FUNCTION_BLOCK FB_BatteryConditioningSFC
VAR_IN_OUT
	IPSDemand					:	ST_PowerDemand;
	ConditioningRequirements	: 	ST_ConditioningRequirements;
	Control						:	ST_CoolingSystem_Control;
	Get							:	ST_CoolingSystemGet;	
END_VAR



VAR_OUTPUT
	SFCCurrentStep	:	STRING;
END_VAR
VAR_OUTPUT
	SFCActive	:	BOOL;
END_VAR

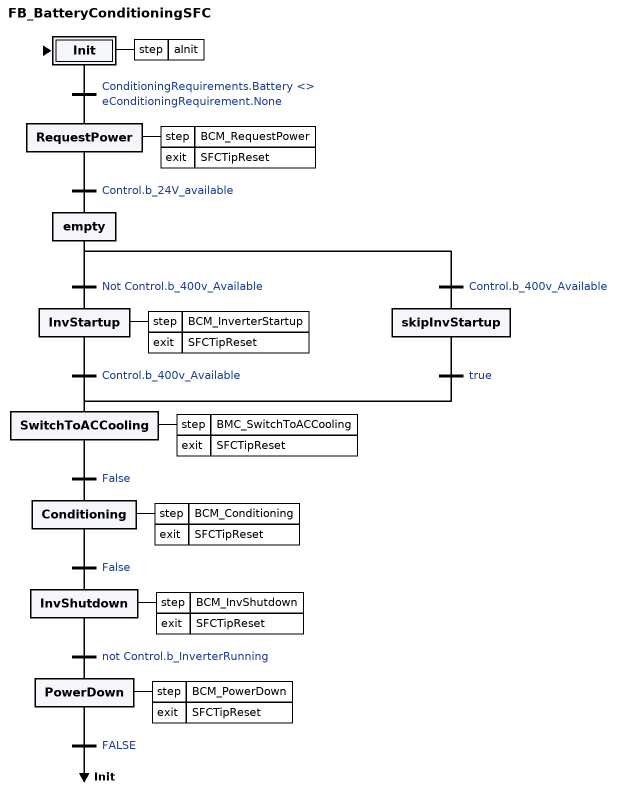
INITIAL_STEP Init:
    aInit(N);  // step action
END_STEP
TRANSITION FROM Init TO RequestPower
    := ConditioningRequirements.Battery <> eConditioningRequirement.None;
END_TRANSITION
STEP RequestPower:
    BCM_RequestPower(N);  // step action
    SFCTipReset(P0);  // exit action
END_STEP
TRANSITION FROM RequestPower TO empty
    := Control.b_24V_available;
END_TRANSITION
STEP empty:
END_STEP
TRANSITION FROM empty TO InvStartup
    := Not Control.b_400v_Available;
END_TRANSITION
STEP InvStartup:
    BCM_InverterStartup(N);  // step action
    SFCTipReset(P0);  // exit action
END_STEP
TRANSITION FROM InvStartup TO SwitchToACCooling
    := Control.b_400v_Available;
END_TRANSITION
TRANSITION FROM empty TO skipInvStartup
    := Control.b_400v_Available;
END_TRANSITION
STEP skipInvStartup:
END_STEP
TRANSITION FROM skipInvStartup TO SwitchToACCooling
    := true;
END_TRANSITION
STEP SwitchToACCooling:
    BMC_SwitchToACCooling(N);  // step action
    SFCTipReset(P0);  // exit action
END_STEP
TRANSITION FROM SwitchToACCooling TO Conditioning
    := False;
END_TRANSITION
STEP Conditioning:
    BCM_Conditioning(N);  // step action
    SFCTipReset(P0);  // exit action
END_STEP
TRANSITION FROM Conditioning TO InvShutdown
    := False;
END_TRANSITION
STEP InvShutdown:
    BCM_InvShutdown(N);  // step action
    SFCTipReset(P0);  // exit action
END_STEP
TRANSITION FROM InvShutdown TO PowerDown
    := not Control.b_InverterRunning;
END_TRANSITION
STEP PowerDown:
    BCM_PowerDown(N);  // step action
    SFCTipReset(P0);  // exit action
END_STEP
TRANSITION FROM PowerDown TO Init
    := FALSE;
END_TRANSITION

ACTION aInit:
SFCActive := False;
END_ACTION

ACTION BCM_Conditioning:

//No real demand for complicated regulation?
//system is off. Just return the average battery temperature to nominal.

//for now just test with fixed setpoints

CASE ConditioningRequirements.Battery OF
	eConditioningRequirement.Cooling:
		Control.e_HeatpumpMode := eHeatpumpmode.Cooling;
		Control.r_HeatPumpSetpoint := 15.0;//minimum adviced battery temperature. Setpoint could be lower, but watch out for inverter condensation.
	eConditioningRequirement.Heating:
		Control.e_HeatpumpMode := eHeatpumpmode.Heating;
		Control.r_HeatPumpSetpoint := 35.0; //minimum heating setpoint
	eConditioningRequirement.None:
		Control.e_HeatpumpMode := eHeatpumpmode.Standby;
		SFCTip := TRUE;
END_CASE

//if coolantpressure drops below startup minimum while inverter is running, shutdown system immediately!
IF 	Control.b_InverterRunning AND
 	(Control.r_CoolantPressure < (CoolingSystemParams.StartupPumpMinimumPressure + Control.r_CoolantIdlePressure)) THEN
		get.Events.b_InverterCoolingLoopError := TRUE;
		ConditioningRequirements.by_PSCoolingPowerMode := 0;
END_IF
END_ACTION

ACTION BCM_Cooldown:

IF ConditioningRequirements.Battery = eConditioningRequirement.Cooling THEN
	Control.b_CloseBatteryLoopValve := FALSE;
	Control.r_HeatPumpSetpoint := 15.0;
ELSIF ConditioningRequirements.Battery = eConditioningRequirement.Heating THEN
	Control.b_CloseBatteryLoopValve := FALSE;
	Control.r_HeatPumpSetpoint := 25.0;
ELSE
	//battery conditioning done, close valve to speed up other conditioning loops
	Control.b_CloseBatteryLoopValve := TRUE;
	IF ConditioningRequirements.Enclosure = eConditioningRequirement.Heating THEN
		Control.r_HeatPumpSetpoint := 25.0;
	ELSIF ConditioningRequirements.Enclosure = eConditioningRequirement.Cooling THEN
		Control.r_HeatPumpSetpoint := 15.0;
	//ELSE
		//if enclosure and battery are ok. Inverter is presumably already cooled down enough. 
		//If not, keep running in current mode for longer
	//	IF PSGet.r_TemperatureMax < CoolingSystemParams.InverterIdleShutdownTemp THEN
		//	ConditioningModeRequired := eConditioningStates.OFF;
		//END_IF
	END_IF	
END_IF
END_ACTION

ACTION BCM_InverterStartup:
Control.b_CloseBatteryLoopValve 	:= TRUE;
Control.b_CloseFancoilLoopValve		:= TRUE;
Control.b_CloseInverterLoopValve	:= FALSE;

Control.b_DCFancoilEnable	:=	FALSE;
//Control.b_ACFancoilEnable	:=	FALSE;

Control.b_DCPumpEnable		:= TRUE;
Control.b_ACPumpEnable		:= FALSE;

Control.b_HeatPumpPowerEnable := FALSE;

//if both are ok, the inverter should have enough flow to start
IF Control.r_CoolantPressure > (CoolingSystemParams.StartupPumpMinimumPressure + Control.r_CoolantIdlePressure) AND Control.b_InverterLoopEnabled THEN
	//Inverter may commence modulating, but no power delivery yet.
	ConditioningRequirements.by_PSCoolingPowerMode := 1;
END_IF
END_ACTION

ACTION BCM_InvShutdown:
Control.b_CloseBatteryLoopValve 	:= TRUE;
Control.b_CloseFancoilLoopValve	:= TRUE;
Control.b_CloseInverterLoopValve	:= FALSE;

Control.b_DCFancoilEnable	:=	FALSE;
//Control.b_ACFancoilEnable	:=	FALSE;

Control.b_DCPumpEnable		:= TRUE;
Control.b_ACPumpEnable		:= FALSE;

Control.b_HeatPumpPowerEnable := FALSE;

//Inverter may shutdown now
ConditioningRequirements.by_PSCoolingPowerMode := 0;
END_ACTION

ACTION BCM_PowerDown:
Control.b_CloseBatteryLoopValve 	:= 	FALSE;
Control.b_CloseFancoilLoopValve	:= 	FALSE;
Control.b_CloseInverterLoopValve	:= 	FALSE;

Control.b_DCFancoilEnable		:=	FALSE;
//Control.b_ACFancoilEnable		:=	FALSE;

Control.b_DCPumpEnable			:= 	FALSE;
Control.b_ACPumpEnable			:= 	FALSE;

Control.b_HeatPumpPowerEnable 	:= 	FALSE;

IPSDemand.b_Demand_24V 			:= FALSE;

Control.e_HeatpumpMode := eHeatpumpMode.Standby; 
SFCActive:= False;
END_ACTION

ACTION BCM_RequestPower:
SFCActive:= True;
IPSDemand.b_Demand_24V := TRUE;
IPSDemand.b_Demand_400V := TRUE;
END_ACTION

ACTION BMC_SwitchToACCooling:
Control.b_DCFancoilEnable 		:= FALSE;
//Control.b_ACFancoilEnable		:= FALSE;


//First enable both pumps to see if AC pump works (by checking pressure increase)
Control.b_ACPumpEnable 			:= TRUE;
Control.b_DCPumpEnable 			:= TRUE;

IF Control.r_CoolantPressure > (CoolingSystemParams.MainPumpMinimumPressure + Control.r_CoolantIdlePressure) THEN
	Control.b_CloseBatteryLoopValve 	:= FALSE;
	Control.b_CloseFancoilLoopValve 	:= FALSE;
	Control.b_CloseBatteryLoopValve 	:= FALSE;
	Control.b_HeatPumpPowerEnable 	:= TRUE;
	Control.b_DCPumpEnable 			:= FALSE;
	Control.e_HeatpumpMode := eHeatpumpmode.Standby;
	Control.r_HeatPumpSetpoint := 18.0;
	SFCTip := TRUE;
END_IF
END_ACTION

METHOD SFCEnable : BOOL
VAR_INPUT
	Enable	:	Bool;
END_VAR
IF Enable THEN
	SFCInit := FALSE;
ELSE
	SFCActive:= FALSE;
	SFCInit := TRUE;
END_IF
END_METHOD

ACTION SFCTipReset:
SFCTip := FALSE;
END_ACTION

END_FUNCTION_BLOCK

(* stored: Version 1.1.0.1, ProductVersion 3.1.4024.12
   POU FB_BatteryConditioningSFC: Id {5ce527d0-615b-41eb-9af7-e543097ab227}, SpecialFunc None
   Action aInit: Id {07ac61e1-8ac9-4677-8bb9-bcdeccba797d}
   Action BCM_Conditioning: Id {4e6a8f50-9ca3-48f3-bb38-f7e201105758}
   Action BCM_Cooldown: Id {466f59fc-3062-467d-b484-59ab2b311a9e}
   Action BCM_InverterStartup: Id {896d08f3-d261-41f2-b071-c750cbf6ce98}
   Action BCM_InvShutdown: Id {2a2e2381-561b-4634-b174-6bb1edc6cb5f}
   Action BCM_PowerDown: Id {3fbcbc49-7065-4971-be73-a2827f1fc09f}
   Action BCM_RequestPower: Id {2758c2a8-6c59-4088-a0e9-6a3d98821783}
   Action BMC_SwitchToACCooling: Id {7a87051e-0eda-454f-98e6-34986fbbb41c}
   Method SFCEnable: Id {d995c454-b52d-4d70-af64-598f34655557}
   Action SFCTipReset: Id {d64fec77-d1a9-4430-83a2-2b9fc1aa4ab1} *)
